TYPE ST_AX5kOut :
STRUCT
	TorquePos  :UINT;		(* =%*30*)
	TorqueNeg :UINT;			(* =%*30*)
END_STRUCT
END_TYPE

(* stored: Version 1.1.0.1, ProductVersion 3.1.4024.11
   DUT ST_AX5kOut: Id {489a8d06-c04c-48a8-8970-0d69291520fb} *)
